TYPE ST_StatusShellyOnePM :
STRUCT

	iOutput					: INT; // -1..status not set, 0..output = false, 1..output = true	

END_STRUCT
END_TYPE

(* stored: Version 1.1.0.1, ProductVersion 3.1.4024.12
   DUT ST_StatusShellyOnePM: Id {5c1c6952-2a97-44f0-93ec-7007955dab58} *)
